FUNCTION_BLOCK Closed
VAR_INPUT
	Enable: BOOL;
	KpGain: LREAL;
	PosRef: LREAL;
	Pos_feedback: LREAL;
END_VAR
VAR_OUTPUT
	Ctrl_signal_Pos: LREAL;
	PosErr: LREAL;
END_VAR
VAR
END_VAR


(* Outputs for Atomic SubSystem: '<Root>/Closed-loop PosCtrl (Auto)' *)
(* Sum: '<S1>/Sum' *)
PosErr := PosRef - Pos_feedback;
(* Product: '<S1>/Product' *)
Ctrl_signal_Pos := KpGain * PosErr;
(* Saturate: '<S1>/Predefined Saturation' *)

IF Ctrl_signal_Pos > 1.0 THEN 
    Ctrl_signal_Pos := 1.0;
ELSIF Ctrl_signal_Pos < -1.0 THEN 
    Ctrl_signal_Pos := -1.0;
END_IF;

(* End of Saturate: '<S1>/Predefined Saturation' *)


(* Switch: '<S1>/Switch' *)

IF Enable := FALSE THEN 
    (* Outport: '<Root>/Ctrl_signal_Pos' incorporates:
     *  Constant: '<S1>/Constant' *)
    Ctrl_signal_Pos := 0.0;
END_IF;

(* End of Switch: '<S1>/Switch' *)
(* End of Outputs for SubSystem: '<Root>/Closed-loop PosCtrl (Auto)' *)

END_FUNCTION_BLOCK

(* stored: Version 1.1.0.1, ProductVersion 3.1.4024.12
   POU Closed: Id {eb4df716-16f4-40fd-ad7a-68452101a208}, SpecialFunc None *)
